FUNCTION LeftArmWristIK : REAL
VAR_INPUT
	theta1:LREAL;					// 左臂右电机角度
	theta2:LREAL;					// 左臂左电机角度
END_VAR
VAR
	// 中间变量
	theta1_rad:LREAL;
	theta2_rad:LREAL;
	rr:LREAL;						//r变量被倍福占用了，所以此处用rr
	u:LREAL;
	angle_ACD:LREAL;
	angle_DCE:LREAL;
	angle_ACE:LREAL;
	angle_ECG:LREAL;
	angle_ECI:LREAL;
	
	point_E:Points;
	point_F:Points;
	
	jx:REAL;				//EF向量的横坐标
	jy:REAL;				//EF向量的纵坐标
	vx:REAL:=0;				//+y单位向量的横坐标
	vy:REAL:=1;				//+y单位向量的纵坐标
	result_cross:REAL;		//EF向量和+y向量的叉乘结果
	
	angle_Beta:REAL;
	
	
END_VAR

theta1_rad := DEG_TO_RAD(theta1);
theta2_rad := DEG_TO_RAD(theta2);

point_F := LeftArmFK(theta1, theta2);

rr := SQRT(EXPT((2*LeftArm_w+LeftArm_f*COS(theta1_rad)-LeftArm_g*COS(theta2_rad)),2) + EXPT((LeftArm_f*SIN(theta1_rad)-LeftArm_g*SIN(theta2_rad)),2));  

u := SQRT(EXPT((2*LeftArm_w-LeftArm_g*COS(theta2_rad)),2) + EXPT((-LeftArm_g*SIN(theta2_rad)),2));

angle_ACD := ACOS((rr*rr+LeftArm_f*LeftArm_f-u*u)/(2*rr*LeftArm_f));

angle_DCE := ACOS((rr*rr + LeftArm_i*LeftArm_i -LeftArm_h*LeftArm_h)/(2*rr*LeftArm_i));

angle_ACE := angle_ACD + angle_DCE;

angle_ECG := angle_ACE - theta1_rad;
    
angle_ECI := PI - angle_ECG;

point_E.x := LeftArm_w + LeftArm_f*COS(theta1_rad) + LeftArm_i*COS(angle_ECI);
point_E.y := LeftArm_f*SIN(theta1_rad) + LeftArm_i*SIN(angle_ECI);

jx := point_F.x - point_E.x;
jy := point_F.y - point_E.y;

result_cross := jx*vy - jy*vx;

IF result_cross > 0 THEN
	angle_Beta := ACOS((jx*vx+jy*vy)/(SQRT(jx*jx+jy*jy)*SQRT(vx*vx+vy*vy)));
ELSIF result_cross < 0 THEN
	angle_Beta := -ACOS((jx*vx+jy*vy)/(SQRT(jx*jx+jy*jy)*SQRT(vx*vx+vy*vy)));
ELSE
	angle_Beta := 0;
END_IF

LeftArmWristIK := RAD_TO_DEG(angle_Beta);

END_FUNCTION

(* stored: Version 1.1.0.1, ProductVersion 3.1.4024.14
   POU LeftArmWristIK: Id {8ee3b6f6-a74e-422b-af29-e9a006f70863}, SpecialFunc None *)
